ABB RobotStudio station: RobotcellV6.rsstn

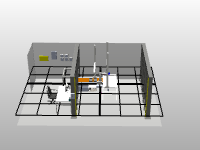
Station RobotcellV6 (saved by RobotStudio 6.7.7936.1011)
Controller MTRN4230
  mechanical unit ROB_1: IRB120_3_58__01, 6 joints, base frame (0, 0, 564.29) mm
Layout (positions relative to the parent item):
  - IRB120_3_58__01 [mechanism, from Robots\IRB120_3_58_G_01.rslib] at (0, 0, 600) mm; joint values [0.0262, 0.0254, -0.0192, -0.0178, -0.0723, 0.7854] (rad or m)
  - Conveyor [part] at (480, 730, 470) mm, rotated rx 90 ry 0 rz 180 deg
  - ConveyorGuard [part] at (-2042, 900, 0) mm, rotated rx 90 ry 0 rz -90 deg
  - CameraFrame [part] at (880, -700, 786) mm, rotated rx 90 ry 0 rz 90 deg
  - TableFrame [part] at (129, 800, 0) mm, rotated rx 90 ry 0 rz -90 deg
  - ConveyorFrame [part] at (200, -716, 600) mm, rotated rx 90 ry 0 rz 90 deg
  - WallGlassLeft [part] at (2500, -2280, 0) mm, rotated rx 90 ry 0 rz 90 deg
  - Box1 [part] at (-190, 200, 600) mm, rotated rx 90 ry 0 rz 90 deg
  - Box2 [part] at (-250, 740, 0) mm
  - TableComputer [part] at (-1300, -1300, 0) mm
  - IRC5_Compact [part, from Equipment\IRC5_Compact.rslib] at (-671.71, 166, 0) mm
  - WalGlasslRight [part] at (-1400, -2250, 0) mm, rotated rx 90 ry 0 rz 90 deg
  - ConveyorControl [part] at (-2800, 1600, 1800) mm, rotated rx 0 ry 90 rz -180 deg
  - PadlockSwitch [part] at (-2300, 1600, 1200) mm, rotated rx 180 ry 0 rz 0 deg
  - PadlockSwitch2 [part] at (-4150, 0, -100) mm
  - PadlockSwitch3 [part] at (-3650, 0, -100) mm
  - PadlockSwitch4 [part] at (0, 0, 2920) mm
  - PadlockSwitch5 [part] at (250, 0, 3063) mm
  - LightCurtainBox [part] at (-3500, 1600, 1200) mm, rotated rx 180 ry 0 rz 0 deg
  - User Library-OFFICE CHAIR [part] at (-2500, -1000, 0) mm, rotated rx 0 ry 0 rz 90 deg
  - User Library-Emergency Stop Switch-2 [part] at (-1187, -700, 1300) mm, rotated rx 90 ry 0 rz 90 deg
  - SafetySwitch [part] at (-1200, -2260, 1100) mm, rotated rx 0 ry -90 rz -180 deg
  - WallLeft [part] at (2500, -2260, 0) mm, rotated rx 90 ry 0 rz 90 deg
  - WallsRight [part] at (-1200, -2257, 0) mm, rotated rx 90 ry 0 rz 90 deg
  - LightCurtainLT [part] at (2260, -2310, 700) mm, rotated rx 90 ry 0 rz 0 deg
  - LightCurtainLB [part] at (2260, -2232, 0) mm, rotated rx 90 ry 0 rz 0 deg
  - LightCurtainRB [part] at (1100, 0, 0) mm
  - LightCurtainRT [part] at (1100, 0, 0) mm
  - User Library-17In Flat Screen-1 [part] at (-1600, -1000, 747) mm, rotated rx 90 ry 0 rz -90 deg
  - ConveyorFrame_2 [part] at (-50, 730, 600) mm, rotated rx 90 ry 0 rz -90 deg
  - PlasticWall [part] at (-1500, 1600, 0) mm, rotated rx 90 ry 0 rz 0 deg
  - Walls_2 [part] at (-2858, 1625, 0) mm, rotated rx 90 ry 0 rz 0 deg
  - Wallss [part] at (-3836, 1625, 0) mm, rotated rx 90 ry 0 rz 0 deg
  - FlexPendant [part, from Equipment\FlexPendant.rslib] at (-1469, -2145, 976) mm, rotated rx 0 ry 0 rz -90 deg
  - Walls_2 [part] at (-3850, 42, 0) mm, rotated rx 90 ry 0 rz 90 deg
  - User Library-Emergency Stop Switch-2 [part] at (-1375.78, 28, 1306) mm, rotated rx 90 ry 0 rz -90 deg
  - WorldFrame [frame]
  - ConveyorFrame [frame] at (0, 409, 622) mm
  - TableFrame [frame] at (175, 0, 747) mm
Targets, tools, work objects and paths stored in the station, written as RAPID:
! task T_ROB1
MODULE Module1
  PROC main()
  ENDPROC
ENDMODULE

! task T_ROB1
MODULE MTRN4230_Server_Sample
  PROC CloseConnection()
  ENDPROC
  PROC MainServer()
  ENDPROC
  PROC ListenForAndAcceptConnection()
  ENDPROC
ENDMODULE

! task T_ROB1
MODULE MTRN4230_IO_Sample
  PROC MainIO()
    WaitTime 2;
    WaitTime 2;
  ENDPROC
  PROC TurnVacOff()
    SetDO DO10_1,0;
  ENDPROC
  PROC TurnConOff()
    SetDO DO10_3,0;
  ENDPROC
  PROC TurnVacOn()
    SetDO DO10_1,1;
  ENDPROC
  PROC TurnConOnSafely()
    SetDO DO10_3,1;
    SetDO DO10_3,0;
  ENDPROC
ENDMODULE

! task T_ROB1
MODULE MTRN4230_Move_Sample
  PROC MoveJSample()
  ENDPROC
  PROC MoveLSample()
    MoveL Offs(pTableHome, 0, 0, 100),v100,fine,tSCup;
  ENDPROC
  PROC MainMove()
    MoveJSample;
    MoveLSample;
  ENDPROC
ENDMODULE

! task T_ROB1
MODULE MTRN4230_IO_Sample
  PROC Main()
    MainIO;
  ENDPROC
  PROC MainIO()
    TurnVacOn;
    WaitTime 2;
    TurnVacOff;
    TurnConOnSafely;
    WaitTime 2;
    TurnConOff;
  ENDPROC
  PROC TurnVacOff()
    SetDO DO10_1,0;
  ENDPROC
  PROC TurnConOff()
    SetDO DO10_3,0;
  ENDPROC
  PROC TurnVacOn()
    SetDO DO10_1,1;
  ENDPROC
  PROC TurnConOnSafely()
    SetDO DO10_3,1;
    SetDO DO10_3,0;
  ENDPROC
ENDMODULE

! task T_ROB1
MODULE MTRN_Rob_Data
  PERS tooldata tSCup:=[TRUE,[[0,0,65],[1,0,0,0]],[0.5,[0,0,20],[1,0,0,0],0,0,0]];
ENDMODULE

